FUNCTION_BLOCK FB_Axis_VirtualSlit EXTENDS FB_Axis
VAR_INPUT
END_VAR
VAR_OUTPUT
END_VAR
VAR
END_VAR

METHOD mControl_LimitLinking : BOOL
//Remove linking of stInput Limits to bFwEnabled and bBwEnabled
_stAxis.stStatus.bInterlockedFwd := _stAxis.stControl.bInterlockFwd;
_stAxis.stStatus.bInterlockedBwd := _stAxis.stControl.bInterlockBwd;

//Multimaster limit linking
FOR nAxisIndex := 1 TO GVL_APP.nAXIS_NUM DO
    IF (_stAxis.stConfig.afMultiSlaveAxisRatio[nAxisIndex] <> 0) THEN
        _stAxis.stStatus.bFwEnabled := _stAxis.stStatus.bFwEnabled AND SEL(_stAxis.stConfig.afMultiSlaveAxisRatio[nAxisIndex] > 0, GVL.astAxes[nAxisIndex].stStatus.bBwEnabled, GVL.astAxes[nAxisIndex].stStatus.bFwEnabled);
        _stAxis.stStatus.bBwEnabled := _stAxis.stStatus.bBwEnabled AND SEL(_stAxis.stConfig.afMultiSlaveAxisRatio[nAxisIndex] > 0, GVL.astAxes[nAxisIndex].stStatus.bFwEnabled, GVL.astAxes[nAxisIndex].stStatus.bBwEnabled);
    END_IF
END_FOR
END_METHOD

METHOD mControl_Power : ST_McStatus
//Change fbPower Enable_Negative and Enable_Positive to monitor stInput limits rather than Bw/Fw Enabled
fbPower.Enable := _stAxis.stControl.bEnable;
fbPower.Enable_Negative := (_stAxis.stInputs.bLimitBwd OR bWaitForStopAfterLimitHit) AND NOT _stAxis.stStatus.bInterlockedBwd;
fbPower.Enable_Positive := (_stAxis.stInputs.bLimitFwd OR bWaitForStopAfterLimitHit) AND NOT _stAxis.stStatus.bInterlockedFwd;
fbPower.Override := _stAxis.stConfig.fOverride;

fbPower(Axis := _stAxis.Axis);

mControl_Power.Error := fbPower.Error;

IF fbPower.Error THEN
    _stAxis.stError.nPowerErrorID := fbPower.ErrorID; //Set the error
END_IF
END_METHOD

END_FUNCTION_BLOCK

(* stored: Version 1.1.0.1, ProductVersion 3.1.4024.11
   POU FB_Axis_VirtualSlit: Id {e31f5dba-ed6e-424e-a71c-5be6f81b1629}, SpecialFunc None
   Method mControl_LimitLinking: Id {8a071033-216a-465d-8f56-bfe7ac105f0a}
   Method mControl_Power: Id {d0c8540c-f48a-44ed-9cab-a42fb64b8fc2} *)
